# EPICS substitutions: MKS660.substitutions
file MKS660.template
{
pattern {S, TA, DN}
	{BL11A, SE, MKS660}
}
